// Mitsubishi GX Works2 project: TestServo   PLC: FX3U/FX3UC

PROGRAM MAIN
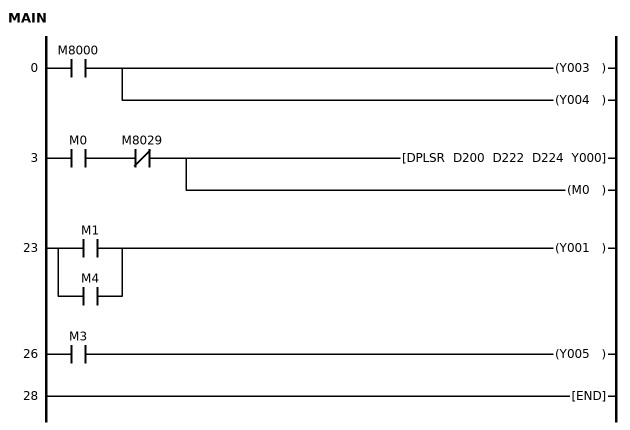
0     LD      M8000
      OUT     Y003
      OUT     Y004
3     LD      M0
      ANI     M8029
      DPLSR   D200 D222 D224 Y000
      OUT     M0
23    LD      M1
      OR      M4
      OUT     Y001
26    LD      M3
      OUT     Y005
28    END
END_PROGRAM
